PROGRAM A_1_PRG_Main_Master
VAR
	
	rtrigButton             				: ARRAY[1..3] OF Tc2_Standard.R_TRIG;
	ftrigButton             				: ARRAY[1..3] OF Tc2_Standard.F_TRIG; 
	
	fbStringFormatter       				: Tc2_Utilities.FB_FormatString;
	fbEventsManager							: FB_EventsManager;
	
	ntShutdown								: TC2_Utilities.NT_Shutdown;
	closeChrome 							: NT_StartProcess;
	tonUserLogOut							: TON;
	fbUserLog								: FB_UserLog;
	
	nFindAdm								: INT;
	nFindEng								: INT;
	nFindOpe								: INT;
	sUserGroupName							: STRING (255);
	sAdmGroup								: STRING (255)							:= 'Administrator';
	sEngGroup								: STRING (255)							:= 'Engineer';
	sOpeGroup								: STRING (255)							:= 'Operator';
	
	rEfficency								: STRING(510);
	
	fbSystemTime							: NT_GetTime;
	
////////////////////////////////////////////////////////////////////////////////////CSV////////////////////////////////////////////////////////////////////////////	

	//stEventsCSVProcess						:  ST_CSVProcess;
	//fbWriteDataToCSV_Events					: FB_WriteDataToCSV;
	fbPDFMaker								: FB_PDFMaker;
	stPDFMaker								: ST_PDFMaker;
	i										: DINT;
	

	
END_VAR

/////////////////////////////////////////////////////////////////////////////////////GENERAL/////////////////////////////////////////////////////////////////////////////////////
A_3_PRG_FaultHandling();
a_ACT_ButtonsLamps();
b_ACT_PDFMaker();
d_ACT_ShutdownAndQuit();
e_ACT_UserLog();
f_ACT_TerminalInfo();
g_ACT_Manual();
h_ACT_Statistics();

C_1_PRG_MainHMI();
//D_1_1_PROG_Write_Data_To_CSV();
//D_2_1_PROG_Write_Data_To_CSV();

PRG_Puls();

// System PowerUP CTRL
tonSystemPowerUP(IN:=bSystemPoweringUP, PT:=tSystemPowerUP_Time);
IF tonSystemPowerUP.Q THEN 
bSystemPoweringUP:=FALSE;
END_IF


A_4_PRG_MasterSystemTime();
/////////////////////////////////////////////////////////////////////////////////////STATIONS/////////////////////////////////////////////////////////////////////////////////////

B_1_1_PRG_Master_Station_1(CMD := CMD_Station1);
B_2_1_PRG_Master_Station_2(CMD := CMD_Station2);
B_3_1_PRG_Master_Station_3(CMD := CMD_Station3);

/////////////////////////////////////////////////////////////////////////////////////PROCESS/////////////////////////////////////////////////////////////////////////////////////

A_2_PRG_MachineCtrl();

/////////////////////////////////////////////////////////////////////////////////////EVENT LOG/////////////////////////////////////////////////////////////////////////////////////

fbEventsManager	(			//INPUTS
							bPulse 							:= stPuls.bFlash10Hz, 
							bResetFaults 					:= bResetTest, 
							stStationEvents 				:= stStationEvents,
							sSystemTime						:= sSystemTime,
							sSystemDate						:= sSystemDate,
 							stEventsAssigment				:= stEventsAssigment,
							bDataWritedInCSV				:= stPDFMaker.bDataWrited,
							
							//OUTPUTS
							astActiveEvents 				=> astActiveEvents,
							astEventsHistory				=> astEventsHistory,
							bWriteDataInCSV					=> stPDFMaker.bWriteData,
							nDataHistoryIndex				=> stPDFMaker.nDataHistoryIndex
							);



////////////////////////////////////////////////////////////////////////////////////SYSTEM DATE & TIME/////////////////////////////////////////////////////////////////////////////////////

fbSystemTime( START := stPuls.bFlash10Hz, TIMESTR => stSystemTime);
	

sSystemTime					:= 	CONCAT( STR1 := WORD_TO_STRING(stSystemTime.wHour), STR2 := CONCAT( STR1 := ':', STR2 := 
								CONCAT( STR1 := WORD_TO_STRING(stSystemTime.wMinute), STR2 := 
								CONCAT(STR1 := ':', STR2 := WORD_TO_STRING(stSystemTime.wSecond)))));
								
sSystemDate					:= 	CONCAT( STR1 := WORD_TO_STRING(stSystemTime.wDay), STR2 := 
								CONCAT(STR1 := '/', STR2 := CONCAT(STR1 := WORD_TO_STRING(stSystemTime.wMonth), STR2 := 
								CONCAT(STR1 := '/', STR2 := WORD_TO_STRING(stSystemTime.wYear)))));

ACTION a_ACT_ButtonsLamps:
//===================================================================
stButtonsLamps.bStartButtonFallingEdge 	:= ftrigButton[1].Q ;
stButtonsLamps.bStartButtonRisingEdge 	:= rtrigButton[1].Q ;
stButtonsLamps.bStopButtonFallingEdge 	:= ftrigButton[2].Q ; 
stButtonsLamps.bStopButtonRisingEdge 	:= rtrigButton[2].Q ;  
stButtonsLamps.bResetButtonFallingEdge 	:= ftrigButton[3].Q ;
stButtonsLamps.bResetButtonRisingEdge 	:= rtrigButton[3].Q ;



ftrigButton[1](CLK :=);
rtrigButton[1](CLK						:=);
ftrigButton[2](CLK						:=);
rtrigButton[2](CLK						:=);
ftrigButton[3](CLK	:=bResetTest 		);
rtrigButton[3](CLK						:=);



//GVL_IO.dw_T11_EL2809.qRESETButton_Indicator := stPuls.bFlash2Hz AND (NOT stMachineStatus.bInitialising AND NOT stMachineStatus.bAutoCycle AND NOT stMachineStatus.bManualMode AND NOT stMachineStatus.bReadyToStart) ;
//GVL_IO.dw_T11_EL2809.qStartButton_Indicator := (stPuls.bFlash2Hz AND stMachineStatus.bReadyToStart) OR (stMachineStatus.bManualMode AND stPuls.bFlash4Hz ) ;
END_ACTION

ACTION b_ACT_PDFMaker:
//EVENTS TO CSV

fbPDFMaker(					
							aDataHistory				:= astEventsHistory,
							bWriteData					:= stPDFMaker.bWriteData,
							sDate						:= stPDFMaker.sDate,
							aDataHistoryArrayLength		:= 1000,
							nDataHistoryIndex			:= stPDFMaker.nDataHistoryIndex,
							sUser						:= 'sebastian',//sUserName,
							sGroup						:= 'administrator',//sUserGroupOut,
							sMachineName				:= 'example',
							
							bDataWrited					=> stPDFMaker.bDataWrited,
							stJavasCriptPDF				=> stJavasCriptPDF,
							bMakePdf					=> stJavasCriptPDF.bMakePDF
							);

(*stPDFMaker.sDate			:= 	CONCAT( STR1 := WORD_TO_STRING(stSystemTime.wDay), STR2 := 
								CONCAT(STR1 := '_', STR2 := CONCAT(STR1 := WORD_TO_STRING(stSystemTime.wMonth), STR2 := 
								CONCAT(STR1 := '_', STR2 := WORD_TO_STRING(stSystemTime.wYear)))));	*)
//CSV
(*fbWriteDataToCSV_Events( 	bWriteData					:= stEventsCSVProcess.bWriteData,
							sFileNamePath				:= stEventsCSVProcess.sFileNamePath,
							sDate						:= stEventsCSVProcess.sDate,
							aDataHistoryArrayLength		:= stEventsCSVProcess.aDataHistoryArrayLength,
							nMAX_CSV_ROWS				:= stEventsCSVProcess.nMAX_CSV_ROWS,
							nMAX_CSV_COLUMNS			:= stEventsCSVProcess.nMAX_CSV_COLUMNS,
							nDataHistoryIndex			:= stEventsCSVProcess.nDataHistoryIndex,
							
							bBusy						=> stEventsCSVProcess.bBusy,
							bError						=> stEventsCSVProcess.bError,
							nErrId						=>,
							bDataWrited					=> stEventsCSVProcess.bDataWrited,
							aDataHistory				:= astEventsHistory);
							

(*stEventsCSVProcess.sDate	:= 	CONCAT( STR1 := WORD_TO_STRING(stSystemTime.wDay), STR2 := 
								CONCAT(STR1 := '_', STR2 := CONCAT(STR1 := WORD_TO_STRING(stSystemTime.wMonth), STR2 := 
								CONCAT(STR1 := '_', STR2 := WORD_TO_STRING(stSystemTime.wYear)))));		*)				
								

stEventsCSVProcess.sFileNamePath						:= 'C:\Users\Sebastian.Ulloa\Desktop\GIT PROJECTS\TEMPLATES\TEMPLATE_VER1\CSV\EVENTS\';								
stEventsCSVProcess.aDataHistoryArrayLength				:= 200;
stEventsCSVProcess.nMAX_CSV_ROWS						:= 1000;
stEventsCSVProcess.nMAX_CSV_COLUMNS						:= 4;*)
END_ACTION

ACTION d_ACT_ShutdownAndQuit:
closeChrome(
    NetId := '',
    PathStr := 'C:\Windows\System32\mshta vbscript:Execute("CreateObject(""WScript.Shell"").Run ""powershell -c',
    DirName := 'C:\Windows\System32\WindowsPowerShell\v1.0',
    ComndLine := 'taskkill /F /IM chrome.exe /T"", 0: window.close")',
    Start := bQuitHmi,
    TmOut := DEFAULT_ADS_TIMEOUT
);
 
bQuitHmi:= FALSE;

ntShutdown(NETID := NetAmsId, DELAY := 5, START := bShutDown);
END_ACTION

ACTION e_ACT_UserLog:
sUserGroupName																:= sUserGroupIn;

nFindAdm	:= TC2_Utilities.FIND( 	STR1									:= sUserGroupName,
									STR2									:= sAdmGroup);
									
nFindEng	:= TC2_Utilities.FIND( 	STR1									:= sUserGroupName,
									STR2									:= sEngGroup);
					
nFindOpe	:= TC2_Utilities.FIND( 	STR1									:= sUserGroupName,
									STR2									:= sOpeGroup);
				
IF nFindAdm <> 0 THEN
	sUserGroupOut															:= 'Administrator';
ELSIF nFindEng <> 0 THEN
	sUserGroupOut															:= 'Engineer';
ELSIF nFindOpe <> 0 THEN
	sUserGroupOut															:= 'Operator';
ELSE sUserGroupOut															:= '';
END_IF

tonUserLogOut( IN := (sUserGroupOut <> 'Administrator' OR sUserGroupOut <> 'Engineer') AND bUserLoggedIn , PT := T#10M);

IF tonUserLogOut.Q THEN
	bLogOut 											:= TRUE;
ELSE bLogOut 											:= FALSE;
END_IF

rUserLoggedIn( CLK := bUserLoggedIn);

fbUserLog(	nNumberOfData								:= 250,
			bSaveSignal									:= rUserLoggedIn.Q, 
			sUser										:= sUserName,
			sGroup										:= sUserGroupOut,
			sDate										:= sSystemDate,
			sTime										:= sSystemTime,
			aDataOutput									:= stUserLog);
END_ACTION

ACTION f_ACT_TerminalInfo:
dw_T03_EL1809.stTerminalInfo.fbTerminalInfo( 	nTerminalState						:= dw_T03_EL1809.stTerminalInfo.nTerminal_State,
												sTerminalState						=> dw_T03_EL1809.stTerminalInfo.sTerminalInfo);
												
dw_T04_EL2809.stTerminalInfo.fbTerminalInfo(	nTerminalState						:= dw_T04_EL2809.stTerminalInfo.nTerminal_State,
												sTerminalState						=> dw_T04_EL2809.stTerminalInfo.sTerminalInfo);
END_ACTION

ACTION g_ACT_Manual:


IF stMachineStatus.bReadyToStart THEN
	bEnableManual											:= TRUE;
ELSE bEnableManual											:= FALSE;
END_IF

IF nMainRegion = 5 AND stMasterCtrl.bNoImmediateFault AND stMasterCtrl.bNoCycleStopFault
	AND NOT stMasterCtrl.bCycleStopRequest AND NOT stButtonsLamps.bStopButtonFallingEdge THEN
	stMasterCtrl.bManualModeRequest							:= TRUE;
	bManualModeOffFlag										:= FALSE;
ELSE 
	stMasterCtrl.bManualModeRequest							:= FALSE; 
	bManualModeOffFlag										:= TRUE;											
END_IF
END_ACTION

ACTION h_ACT_Statistics:
stStatisticsHMI[0].sName			:= 'TOTAL';

stStatisticsHMI[0].nGood		:= stStatisticsHMI[1].nGood + stStatisticsHMI[2].nGood + stStatisticsHMI[3].nGood;
stStatisticsHMI[0].nTotalGood	:= stStatisticsHMI[1].nTotalGood + stStatisticsHMI[2].nTotalGood + stStatisticsHMI[3].nTotalGood;
stStatisticsHMI[0].nBad			:= stStatisticsHMI[1].nBad + stStatisticsHMI[2].nBad + stStatisticsHMI[3].nBad;
stStatisticsHMI[0].nTotalBad	:= stStatisticsHMI[1].nTotalBad + stStatisticsHMI[2].nTotalBad + stStatisticsHMI[3].nTotalBad;

								

IF (( stStatisticsHMI[0].nGood + stStatisticsHMI[0].nBad) <> 0) THEN
	
	rEfficency							:= LREAL_TO_FMTSTR(in := (DINT_TO_REAL(stStatisticsHMI[0].nGood) /( DINT_TO_REAL(stStatisticsHMI[0].nGood) + DINT_TO_REAL(stStatisticsHMI[0].nBad))) * 100.0,iPrecision := 2, bRound := TRUE);
	stStatisticsHMI[0].nEfficency		:= CONCAT(STR1 := '%', STR2 := (rEfficency));

ELSE stStatisticsHMI[0].nEfficency		:= CONCAT(STR1 := '%', STR2 := (DINT_TO_STRING(0)));
	
END_IF
END_ACTION

END_PROGRAM

(* stored: Version 1.1.0.1, ProductVersion 3.1.4024.13
   POU A_1_PRG_Main_Master: Id {f5cadd41-0b0d-4992-977e-5b237965be89}, SpecialFunc None
   Action a_ACT_ButtonsLamps: Id {bc3442d0-b536-4f84-a62c-f220009c35e9}
   Action b_ACT_PDFMaker: Id {eda48c17-c939-4052-a903-aa51ced32374}
   Action d_ACT_ShutdownAndQuit: Id {b7dac9a1-fefc-426e-a57f-b21e21205edc}
   Action e_ACT_UserLog: Id {804f315c-0a35-4a48-b9b3-6593241a417c}
   Action f_ACT_TerminalInfo: Id {8299d142-9ce5-4d1b-9f3f-121127d1dbfb}
   Action g_ACT_Manual: Id {87b8b019-9eb6-46b9-b781-3301c89600c8}
   Action h_ACT_Statistics: Id {00b1c5d7-138a-4e5a-aad9-c5f6ae987c75} *)
